FUNCTION_BLOCK CrossJoystick (* Joystick block with 4 directional states and Center, transitions only over Center *)
  (* Standard: 61499-2 *)
  (* Version 1.0, 2026-06-12, Franz Höpfinger *)
  PACKAGE MyLib::sys;
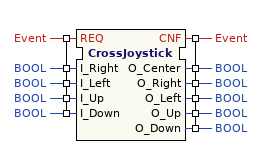
  EVENT_INPUT
    REQ WITH I_Right, I_Left, I_Up, I_Down; (* Update State *)
  END_EVENT
  EVENT_OUTPUT
    CNF WITH O_Center, O_Right, O_Left, O_Up, O_Down; (* State Updated *)
  END_EVENT
  VAR_INPUT
    I_Right : BOOL := FALSE; (* Right Input *)
    I_Left : BOOL := FALSE; (* Left Input *)
    I_Up : BOOL := FALSE; (* Up Input *)
    I_Down : BOOL := FALSE; (* Down Input *)
  END_VAR
  VAR_OUTPUT
    O_Center : BOOL := TRUE; (* Center Output *)
    O_Right : BOOL := FALSE; (* Right Output *)
    O_Left : BOOL := FALSE; (* Left Output *)
    O_Up : BOOL := FALSE; (* Up Output *)
    O_Down : BOOL := FALSE; (* Down Output *)
  END_VAR
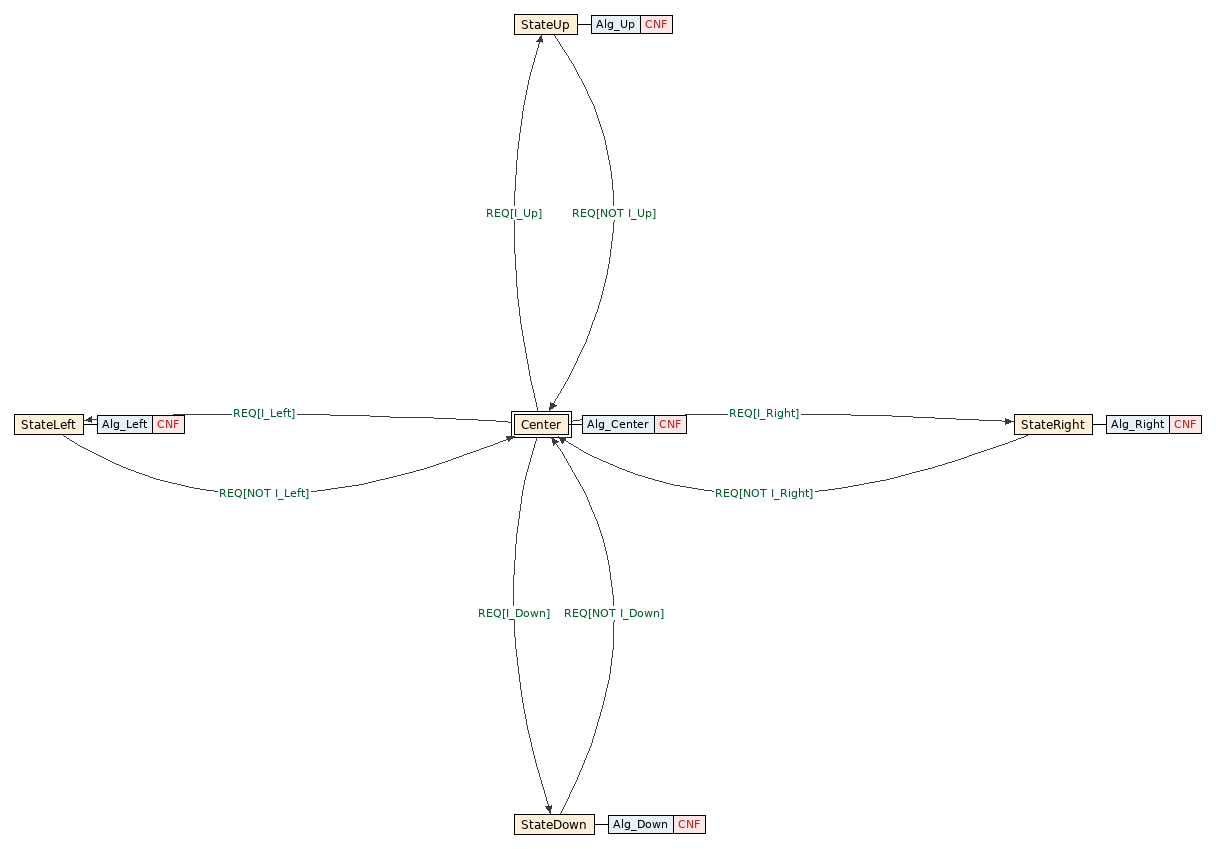
  EC_STATES
    Center : Alg_Center -> CNF; (* Center position *)
    StateRight : Alg_Right -> CNF; (* Right position *)
    StateLeft : Alg_Left -> CNF; (* Left position *)
    StateUp : Alg_Up -> CNF; (* Up position *)
    StateDown : Alg_Down -> CNF; (* Down position *)
  END_STATES
  EC_TRANSITIONS
    Center TO StateRight := REQ[I_Right];
    Center TO StateLeft := REQ[I_Left];
    Center TO StateUp := REQ[I_Up];
    Center TO StateDown := REQ[I_Down];
    StateRight TO Center := REQ[NOT I_Right];
    StateLeft TO Center := REQ[NOT I_Left];
    StateUp TO Center := REQ[NOT I_Up];
    StateDown TO Center := REQ[NOT I_Down];
  END_TRANSITIONS
  ALGORITHM Alg_Center IN ST: (* Center position active *)
O_Center := TRUE;
O_Right := FALSE;
O_Left := FALSE;
O_Up := FALSE;
O_Down := FALSE;
  END_ALGORITHM
  ALGORITHM Alg_Right IN ST: (* Right position active *)
O_Center := FALSE;
O_Right := TRUE;
O_Left := FALSE;
O_Up := FALSE;
O_Down := FALSE;
  END_ALGORITHM
  ALGORITHM Alg_Left IN ST: (* Left position active *)
O_Center := FALSE;
O_Right := FALSE;
O_Left := TRUE;
O_Up := FALSE;
O_Down := FALSE;
  END_ALGORITHM
  ALGORITHM Alg_Up IN ST: (* Up position active *)
O_Center := FALSE;
O_Right := FALSE;
O_Left := FALSE;
O_Up := TRUE;
O_Down := FALSE;
  END_ALGORITHM
  ALGORITHM Alg_Down IN ST: (* Down position active *)
O_Center := FALSE;
O_Right := FALSE;
O_Left := FALSE;
O_Up := FALSE;
O_Down := TRUE;
  END_ALGORITHM
END_FUNCTION_BLOCK
